Staubli VAL3: RobotStatus.dtx

public num nDrivesPowered
public num nEStopped
public num nErrorCode
public num nInError
public num nInMotion
public num nMode
public num nMotionPossible
public num nTrajectoryComplete
